FUNCTION F_BPWithID : ST_BP_ArbInternal
VAR_INPUT
    BP : REFERENCE TO ST_BeamParams;
    ID : DWORD;
END_VAR
VAR
    BpInt : ST_BP_ArbInternal;
END_VAR

MEMCPY(ADR(F_BPWithID), ADR(BP), SIZEOF(BP));
F_BPWithID.nId := ID;

END_FUNCTION

(* stored: Version 1.1.0.1, ProductVersion 3.1.4022.18
   POU F_BPWithID: Id {e3bfa99b-9d0a-4973-9793-594c4c68e1ba}, SpecialFunc None *)
